INTERFACE I_HE_SolidAttenuatorState EXTENDS I_Fallible


METHOD GetState : E_HE_SolidAttenuatorState
END_METHOD

END_INTERFACE

(* stored: Version 1.1.0.1
   Itf I_HE_SolidAttenuatorState: Id {a3e53fae-c57e-4a2e-92e1-c5849e8de238}
   Method GetState: Id {d87b2537-df7d-4545-84af-f73c3719ed51} *)
